// TIA Portal V19 export
DATA_BLOCK "Area03_Messages"   // DB108
// stored: MemoryReserve 100
   VAR
      "A" : Struct
         Msg : Array[1..736] of Bool;
         Hmi : Array[1..46] of Word;
         Ack : Array[1..46] of Word;
      END_STRUCT;
      W : Struct
         Msg : Array[1..832] of Bool;
         Hmi : Array[1..52] of Word;
         Ack : Array[1..52] of Word;
      END_STRUCT;
   END_VAR
BEGIN
   // "A".Msg[2] : h
   // "A".Msg[3] : hsfdd
END_DATA_BLOCK
